FUNCTION_BLOCK SafetyAndOrFB EXTENDS SafetyBase
VAR
END_VAR

METHOD CyclicLogic
VAR_INST
END_VAR
SUPER^.CyclicLogic();
_OK := SUPER^.InfoData.State = E_SafetyOrAnd_State.Run;
END_METHOD

END_FUNCTION_BLOCK

(* stored: Version 1.1.0.1, ProductVersion 3.1.4026.18
   POU SafetyAndOrFB: Id {38938398-edc5-4349-baf8-8c79fa3f2ecf}, SpecialFunc None
   Folder Cyclic: Id {8ca1ae71-ab8e-487f-ac45-f623e9025320}
   Method CyclicLogic: Id {dfb61799-1c78-469c-b931-88ac019768f9} *)
